% RSLogix 500 project Digital Pump Control.RSS, saved by version 8.30.00.16 %
PROJECT "UNTITLED"    % processor: Bul.1763 MicroLogix 1100 Series B %

PROGRAM FILES
  LAD 2 "MAIN"  3 rungs
  LAD 3 "DIGITAL IO"  7 rungs
  LAD 4 "CONTROLS"  6 rungs

DATA FILES
  O0 OUTPUT  5 elements
  I1 INPUT  7 elements
  S2 STATUS  66 elements
  B3 BINARY  1 elements
  T4 TIMER  2 elements
  C5 COUNTER  1 elements
  R6 CONTROL  1 elements
  N7 INTEGER  1 elements
  F8 FLOAT  1 elements

LADDER 2 "MAIN"
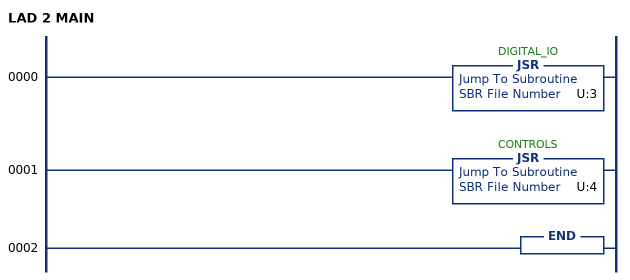
% Rung: 0 %
SOR JSR U:3 EOR
%   U:3  "DIGITAL_IO" %
% Rung: 1 %
SOR JSR U:4 EOR
%   U:4  "CONTROLS" %
% Rung: 2 %
SOR END EOR

LADDER 3 "DIGITAL IO"
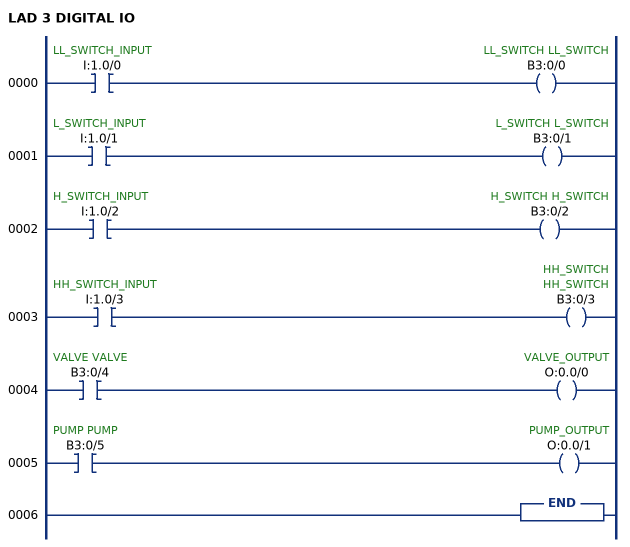
% Rung: 0 %
SOR XIC I:1.0/0 OTE B3:0/0 EOR
%   I:1.0/0  "LL_SWITCH_INPUT" %
%   B3:0/0  LL_SWITCH  "LL_SWITCH" %
% Rung: 1 %
SOR XIC I:1.0/1 OTE B3:0/1 EOR
%   I:1.0/1  "L_SWITCH_INPUT" %
%   B3:0/1  L_SWITCH  "L_SWITCH" %
% Rung: 2 %
SOR XIC I:1.0/2 OTE B3:0/2 EOR
%   I:1.0/2  "H_SWITCH_INPUT" %
%   B3:0/2  H_SWITCH  "H_SWITCH" %
% Rung: 3 %
SOR XIC I:1.0/3 OTE B3:0/3 EOR
%   I:1.0/3  "HH_SWITCH_INPUT" %
%   B3:0/3  HH_SWITCH  "HH_SWITCH" %
% Rung: 4 %
SOR XIC B3:0/4 OTE O:0.0/0 EOR
%   B3:0/4  VALVE  "VALVE" %
%   O:0.0/0  "VALVE_OUTPUT" %
% Rung: 5 %
SOR XIC B3:0/5 OTE O:0.0/1 EOR
%   B3:0/5  PUMP  "PUMP" %
%   O:0.0/1  "PUMP_OUTPUT" %
% Rung: 6 %
SOR END EOR

LADDER 4 "CONTROLS"
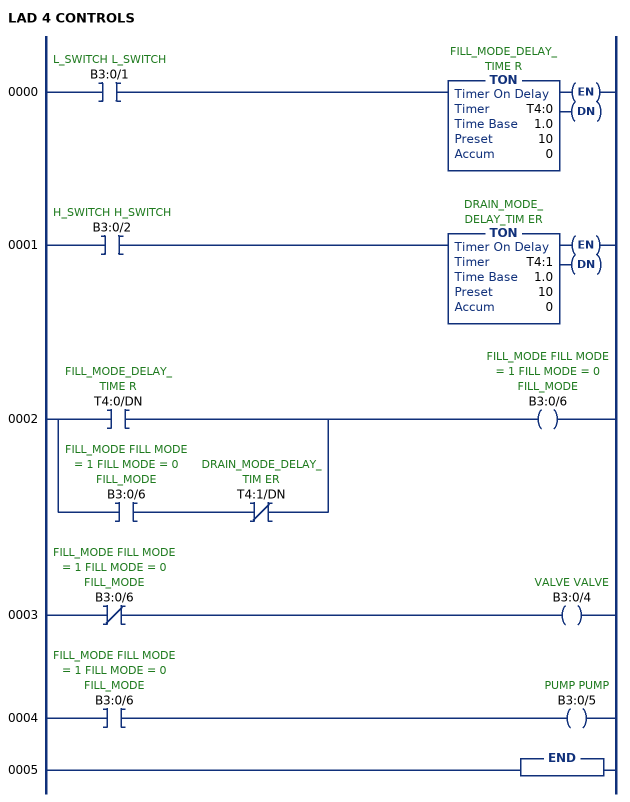
% Rung: 0 %
SOR XIC B3:0/1 TON T4:0 1.0 10 0 EOR
%   B3:0/1  L_SWITCH  "L_SWITCH" %
%   T4:0  "FILL_MODE_DELAY_TIME R" %
% Rung: 1 %
SOR XIC B3:0/2 TON T4:1 1.0 10 0 EOR
%   B3:0/2  H_SWITCH  "H_SWITCH" %
%   T4:1  "DRAIN_MODE_DELAY_TIM ER" %
% Rung: 2 %
SOR BST XIC T4:0/DN NXB XIC B3:0/6 XIO T4:1/DN BND OTE B3:0/6 EOR
%   T4:0  "FILL_MODE_DELAY_TIME R" %
%   B3:0/6  FILL_MODE  "FILL_MODE FILL MODE = 1 FILL MODE = 0" %
%   T4:1  "DRAIN_MODE_DELAY_TIM ER" %
% Rung: 3 %
SOR XIO B3:0/6 OTE B3:0/4 EOR
%   B3:0/6  FILL_MODE  "FILL_MODE FILL MODE = 1 FILL MODE = 0" %
%   B3:0/4  VALVE  "VALVE" %
% Rung: 4 %
SOR XIC B3:0/6 OTE B3:0/5 EOR
%   B3:0/6  FILL_MODE  "FILL_MODE FILL MODE = 1 FILL MODE = 0" %
%   B3:0/5  PUMP  "PUMP" %
% Rung: 5 %
SOR END EOR

OTHER DOCUMENTED ADDRESSES
  O:0  "VALVE_OUTPUT"

DATA TABLE (non-zero values as saved)
DATA T4
% .PRE .ACC %
% T4:0 % 10 0
% T4:1 % 10 0
